# EPICS substitutions: epics_installer_v1.0/option/testIOC/db/user.substitutions
# Example substitutions file

file "db/circle.db" {
    { user = "musr4" }
}

file "db/dbExample1.db" {
    { user = "musr4" }
}

file db/dbExample2.db {
    pattern { user, no, scan }
        { "musr4", 1, "1 second" }
        { "musr4", 2, "2 second" }
        { "musr4", 3, "5 second" }
}
